FUNCTION_BLOCK CM_Actuator3State_V2
VAR_INPUT
	Local_MODE_request : ENUM_MODE_HANDLER;
	Global_MODE_request : ENUM_MODE_HANDLER;
	
	PI_MANUAL :BOOL;
	PI_HMI_HAND : BOOL;
	PI_AUTO : BOOL;
	
	PI_MANUAL_ON_1 : BOOL;
	PI_MANUAL_ON_2 : BOOL;
	
	PI_AUTO_ON_1 : BOOL;
	PI_AUTO_ON_2 : BOOL;
	
	PI_OFF : BOOL;
	
	PI_Alarm_Enable : BOOL;
	PI_CM_Alarm : BOOL;
	
	PI_CM_Interlock : BOOL;
END_VAR
VAR_OUTPUT
	IN_ON : BOOL;
	
	PO_AUTO_ON :BOOL;
	PO_MANUAL_ON :BOOL;
	PO_HMI_HAND_ON : BOOL;
	
	PO_ON_1 : BOOL;
	PO_ON_2 : BOOL;
	
	PO_OFF :BOOL;
	
	PO_CM_Alarm : BOOL;
	
	PO_CM_Interlocked : BOOL;
	
	
END_VAR
VAR
	alarmDelay_H : systemTimeDelay;
	alarmDelay_L : systemTimeDelay;
	
	MODE_HANDLER : FB_MODE_HANDLER;
END_VAR
VAR_IN_OUT
	
END_VAR

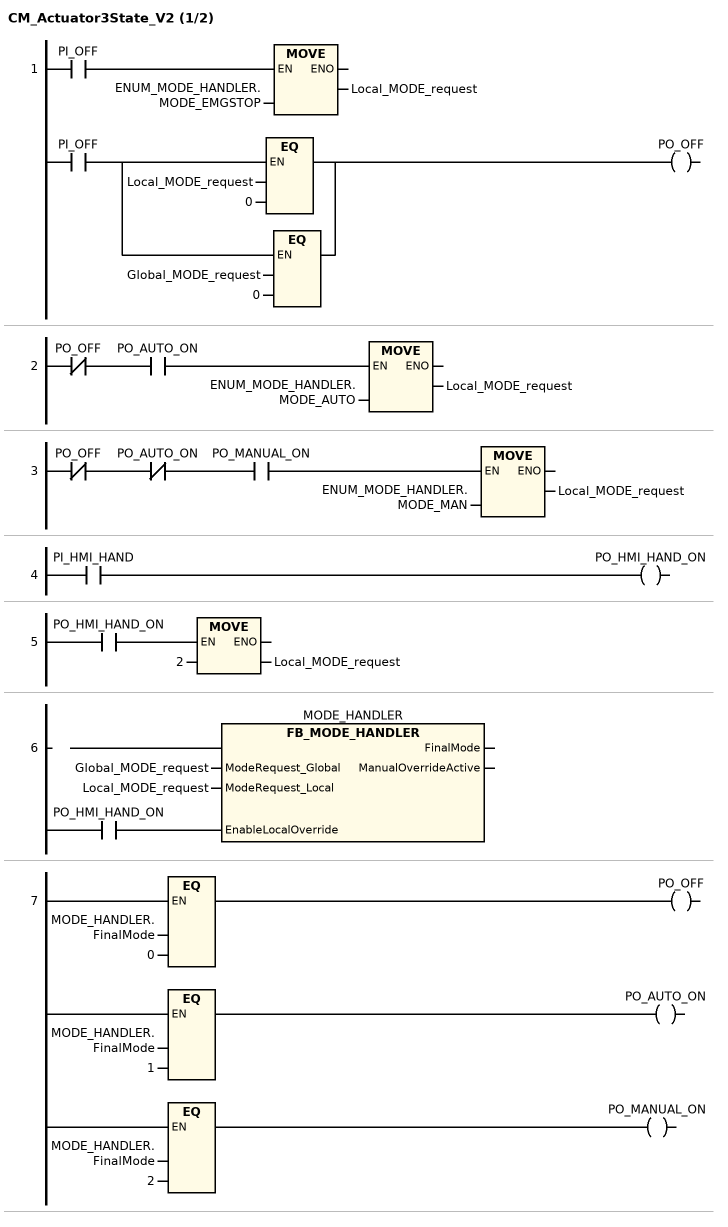
// NETWORK 1
IF PI_OFF THEN Local_MODE_request := ENUM_MODE_HANDLER.MODE_EMGSTOP; END_IF
PO_OFF := PI_OFF AND Local_MODE_request = 0 OR PI_OFF AND Global_MODE_request = 0;

// NETWORK 2
IF NOT PO_OFF AND PO_AUTO_ON THEN Local_MODE_request := ENUM_MODE_HANDLER.MODE_AUTO; END_IF

// NETWORK 3
IF NOT PO_OFF AND NOT PO_AUTO_ON AND PO_MANUAL_ON THEN Local_MODE_request := ENUM_MODE_HANDLER.MODE_MAN; END_IF

// NETWORK 4
PO_HMI_HAND_ON := PI_HMI_HAND;

// NETWORK 5
IF PO_HMI_HAND_ON THEN Local_MODE_request := 2; END_IF

// NETWORK 6
MODE_HANDLER(
    ModeRequest_Global := Global_MODE_request,
    ModeRequest_Local := Local_MODE_request,
    EnableLocalOverride := PO_HMI_HAND_ON); // FB_MODE_HANDLER

// NETWORK 7
PO_OFF := MODE_HANDLER.FinalMode = 0;
PO_AUTO_ON := MODE_HANDLER.FinalMode = 1;
PO_MANUAL_ON := MODE_HANDLER.FinalMode = 2;

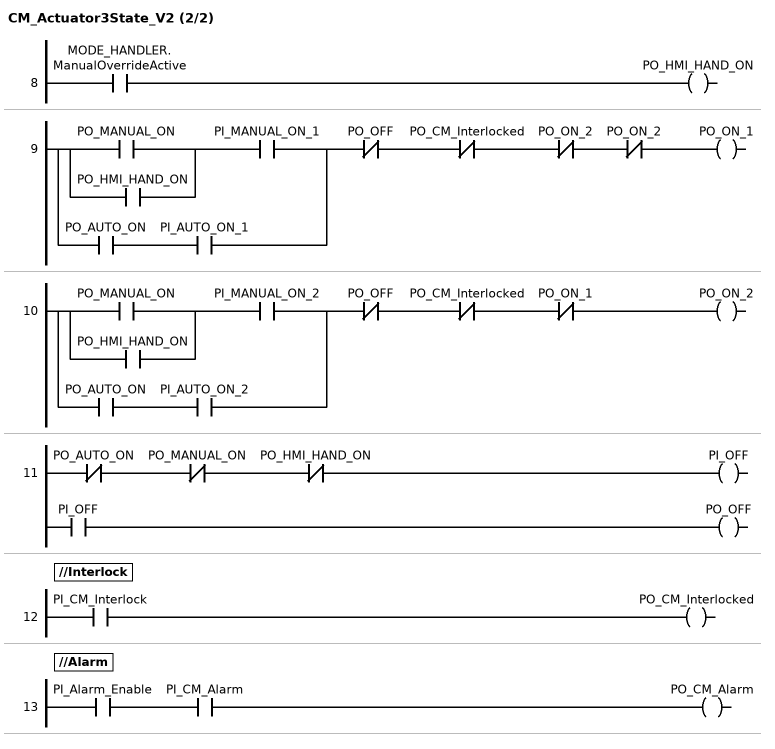
// NETWORK 8
PO_HMI_HAND_ON := MODE_HANDLER.ManualOverrideActive;

// NETWORK 9
PO_ON_1 := ((PO_MANUAL_ON OR PO_HMI_HAND_ON) AND PI_MANUAL_ON_1 OR PO_AUTO_ON AND PI_AUTO_ON_1) AND NOT PO_OFF AND NOT PO_CM_Interlocked AND NOT PO_ON_2 AND NOT PO_ON_2;

// NETWORK 10
PO_ON_2 := ((PO_MANUAL_ON OR PO_HMI_HAND_ON) AND PI_MANUAL_ON_2 OR PO_AUTO_ON AND PI_AUTO_ON_2) AND NOT PO_OFF AND NOT PO_CM_Interlocked AND NOT PO_ON_1;

// NETWORK 11
PI_OFF := NOT PO_AUTO_ON AND NOT PO_MANUAL_ON AND NOT PO_HMI_HAND_ON;
PO_OFF := PI_OFF;

// NETWORK 12
// label: //Interlock
PO_CM_Interlocked := PI_CM_Interlock;

// NETWORK 13
// label: //Alarm
PO_CM_Alarm := PI_Alarm_Enable AND PI_CM_Alarm;

END_FUNCTION_BLOCK

(* stored: Version 1.1.0.1, ProductVersion 3.1.4024.13
   POU CM_Actuator3State_V2: Id {71b2a1ae-eee5-4caf-bbd1-7030f1b44873}, SpecialFunc None *)
